{attribute 'qualified_only'}
VAR_GLOBAL
	Segment	: ARRAY [4..6] OF ST_Segment_Base;
END_VAR

(* stored: Version 1.1.0.1, ProductVersion 3.1.4024.11
   GVL LCP2_IO: Id {3e3a4ec7-086e-46f4-8f09-1c81d482d72e} *)
